% RSLogix 500 project TANK_ANAL_BAK000.RSS, saved by version 8.30.00.16 %
PROJECT "UNTITLED"    % processor: Bul.1763 MicroLogix 1100 Series B %

PROGRAM FILES
  LAD 2 "MAIN"  3 rungs
  LAD 3 "ANALOG IO"  4 rungs
  LAD 4 "CONTROLS"  3 rungs

DATA FILES
  O0 OUTPUT  5 elements
  I1 INPUT  14 elements
  S2 STATUS  66 elements
  B3 BINARY  1 elements
  T4 TIMER  1 elements
  C5 COUNTER  1 elements
  R6 CONTROL  1 elements
  N7 INTEGER  1 elements
  F8 FLOAT  1 elements

LADDER 2 "MAIN"
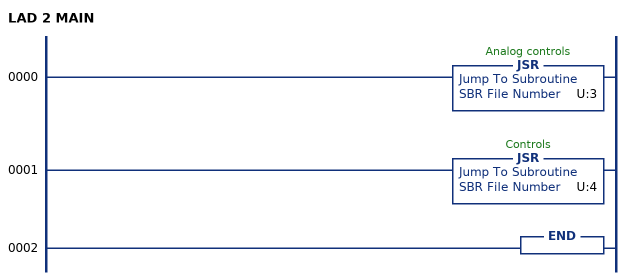
% Rung: 0 %
SOR JSR U:3 EOR
%   U:3  "Analog controls" %
% Rung: 1 %
SOR JSR U:4 EOR
%   U:4  "Controls" %
% Rung: 2 %
SOR END EOR

LADDER 3 "ANALOG IO"
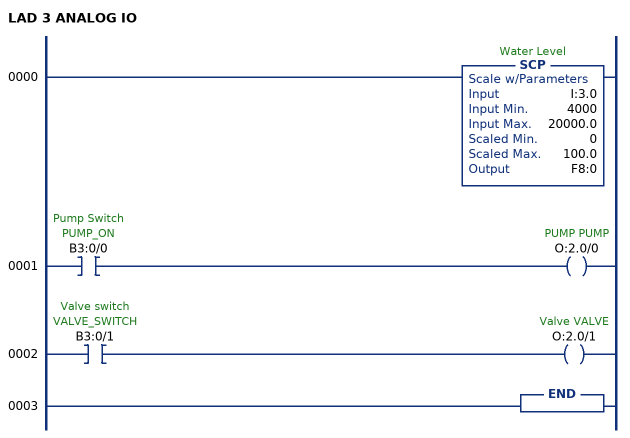
% Rung: 0 %
SOR SCP I:3.0 4000 20000.0 0 100.0 F8:0 EOR
%   I:3.0  WATER_LEVEL  "Water Level" %
%   F8:0  "Water Level" %
% Rung: 1 %
SOR XIC B3:0/0 OTE O:2.0/0 EOR
%   B3:0/0  PUMP_ON  "Pump Switch" %
%   O:2.0/0  PUMP  "PUMP" %
% Rung: 2 %
SOR XIC B3:0/1 OTE O:2.0/1 EOR
%   B3:0/1  VALVE_SWITCH  "Valve switch" %
%   O:2.0/1  VALVE  "Valve" %
% Rung: 3 %
SOR END EOR

LADDER 4 "CONTROLS"
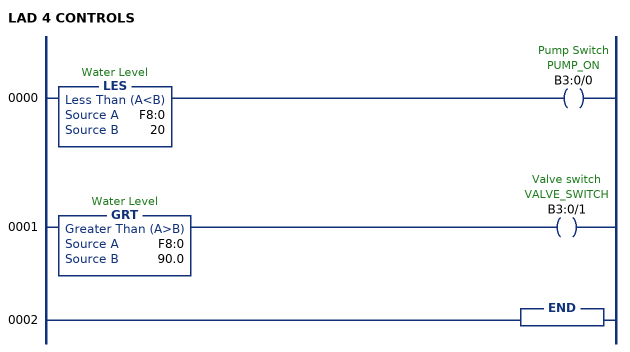
% Rung: 0 %
SOR LES F8:0 20 OTE B3:0/0 EOR
%   F8:0  "Water Level" %
%   B3:0/0  PUMP_ON  "Pump Switch" %
% Rung: 1 %
SOR GRT F8:0 90.0 OTE B3:0/1 EOR
%   F8:0  "Water Level" %
%   B3:0/1  VALVE_SWITCH  "Valve switch" %
% Rung: 2 %
SOR END EOR

OTHER DOCUMENTED ADDRESSES
  O:2.0  "WATER LEVEL OUT"
